// GET THE CURRENT VOLUME OF LIQUID IN THE TANK [m3]

FUNCTION GetVolume : REAL

VAR
	
	a : REAL := tank.A;
	h : REAL := High.now;
	
END_VAR

GetVolume := a * h;

END_FUNCTION

(* stored: Version 1.1.0.1, ProductVersion 3.1.4024.12
   POU GetVolume: Id {77c24618-b925-4840-a558-accae81d177a}, SpecialFunc None *)
